FUNCTION "ST10_Device" : Void
VAR_INPUT
  iSysMode : "RCS_SysComInterface_V1";
END_VAR
BEGIN
  // Původní jazyk: LAD
  // Zdroj XML: EXPORT/Program blocks/OP010/10_Device/ST10_Device.xml
  // (Žádný StructuredText network nebyl nalezen; LAD/STL/GRAPH není automaticky překládán.)
END_FUNCTION
